// TIA Portal V20 export
DATA_BLOCK "CallEquipment_DB"   // DB148
{ DB_Accessible_From_OPC_UA := 'FALSE' }
// stored: AssignedProDiagFB Unit1.Em3.ProDiag, DBAccessibleFromOPCUA false, DBAccessibleFromWebserver false, InstanceOfName Unit1.Em3.CallEquipment, InstanceOfType FB, Namespace Unit1.Em3
"Unit1.Em3.CallEquipment"
   // VAR_INPUT
   //    ZoneOperationEnable { ExternalWritable := 'False'} : "LWONIK_typeSafetyZoneManualOperation";
   // END_VAR
   // VAR_IN_OUT
   //    unitStatus : "LAF_typeUnitStatus";
   //    emFeedback : "LUC_typeEmFeedback";
   //    unitAlarmDB : "LAF_typeAlarms";
   // END_VAR
   // VAR
   //    InstSequenceTopTapeLoading { ExternalWritable := 'False'} : "Unit1.Em3.Sequence_1_TopTapeLoading";
   //    InstSequenceTopTapeAttachment { ExternalWritable := 'False'} : "Unit1.Em3.Sequence_2_TopTapeAttachment";
   //    InstSequenceTopTapeFixStage { ExternalWritable := 'False'} : "Unit1.Em3.Sequence_3_TopTapeFixStage";
   //    instTopTapeLoadingHomeJob1 { ExternalWritable := 'False'} : "LAF_SelectJob";
   //    instTopTapeLoadingChargeJob2 { ExternalWritable := 'False'} : "LAF_SelectJob";
   //    instTopTapeAttachHomeJob1 { ExternalWritable := 'False'} : "LAF_SelectJob";
   //    instTopTapeAttachTapeGetJob2 { ExternalWritable := 'False'} : "LAF_SelectJob";
   //    instTopTapeAttachTape1PutJob3 { ExternalWritable := 'False'} : "LAF_SelectJob";
   //    instTopTapeAttachTape2PutJob4 { ExternalWritable := 'False'} : "LAF_SelectJob";
   //    instTopTapeAttachTapeIdleJob5 { ExternalWritable := 'False'} : "LAF_SelectJob";
   //    instTopTapeFixStageHomeJob1 { ExternalWritable := 'False'} : "LAF_SelectJob";
   //    instTopTapeFixStageLoadJob2 { ExternalWritable := 'False'} : "LAF_SelectJob";
   //    instTopTapeFixStageTaping1Job3 { ExternalWritable := 'False'} : "LAF_SelectJob";
   //    instTopTapeFixStageTaping2Job4 { ExternalWritable := 'False'} : "LAF_SelectJob";
   //    instTopTapeFixStageUnloadJob5 { ExternalWritable := 'False'} : "LAF_SelectJob";
   //    instCmTopTapeJRDetect { ExternalWritable := 'False'} : "LBC_DigitalSignalCn";
   //    instCmTopTapeDiameter { ExternalWritable := 'False'} : "LBC_DigitalSignalCn";
   //    instCmTopTapeAxisX { ExternalWritable := 'False'} : "LBC_Axis64Pos_TecPlcCn";
   //    instCmTopTapeAxisY { ExternalWritable := 'False'} : "LBC_Axis64Pos_TecPlcCn";
   //    instCmTopTapeLoadingFwdBwd { ExternalWritable := 'False'} : "LBC_TwoWayActuatorCn";
   //    instCmTopTapeLoadingClampOpenClose { ExternalWritable := 'False'} : "LBC_TwoWayActuatorCn";
   //    instCmTopTapeCutterUpDown { ExternalWritable := 'False'} : "LBC_TwoWayActuatorCn";
   //    instCmTopTapeCutterClampUpDown { ExternalWritable := 'False'} : "LBC_TwoWayActuatorCn";
   //    instCmTopTapeTensionFwdBwd { ExternalWritable := 'False'} : "LBC_TwoWayActuatorCn";
   //    instCmTopTapeAttachmentUpDown { ExternalWritable := 'False'} : "LBC_TwoWayActuatorCn";
   //    instCmTopTapeClampTopLeftUpDown { ExternalWritable := 'False'} : "LBC_TwoWayActuatorCn";
   //    instCmTopTapeClampTopCenterUpDown { ExternalWritable := 'False'} : "LBC_TwoWayActuatorCn";
   //    instCmTopTapeClampTopRightUpDown { ExternalWritable := 'False'} : "LBC_TwoWayActuatorCn";
   //    instCmTopTapeClampBtmDownUp { ExternalWritable := 'False'} : "LBC_TwoWayActuatorCn";
   //    instCmTopTapeClampAllOpenClose { ExternalWritable := 'False'} : "LBC_TwoWayActuatorCn";
   //    instCmTopTapeAttachmentVaccumOffOn { ExternalWritable := 'False'} : "LBC_TwoWayActuatorCn";
   //    instQrHandyReader { ExternalWritable := 'False'} : "LER_QRread_DM8700";
   //    instInterlockTopTapeAxisX { ExternalWritable := 'False'} : "LER_Axis64Pos_InterlockSummary";
   //    instInterlockTopTapeAxisY { ExternalWritable := 'False'} : "LER_Axis64Pos_InterlockSummary";
   //    instEventsPFE { ExternalWritable := 'False'} : "Unit1.Em3.EventsPFE";
   //    instManageAlarms { ExternalWritable := 'False'} : "LAF_ManageAlarms";
   //    statUnitStatus { ExternalWritable := 'False'} : "LAF_typeUnitStatus";
   //    statSlmStatus { ExternalWritable := 'False'} : Struct
   //       running : Bool;
   //       powerOff : Bool;
   //    END_STRUCT;
   //    statEmptyJobStatus { ExternalWritable := 'False'} : "LAF_typeJobStatus";
   //    statTonTime { ExternalWritable := 'False'} : Array[0..999] of TON_TIME;
   //    statTofTime { ExternalWritable := 'False'} : Array[0..9] of TOF_TIME;
   //    statPulse { ExternalWritable := 'False'} : Array[0..999] of Bool;
   //    statEnableManualCmds { ExternalWritable := 'False'} : Bool;
   //    TopTapeIdleCondition : Bool;
   //    "*** Interlock Axis ***" : Bool;
   //    TopTapeAxisX_JogCW { S7_SetPoint := 'True'} : "LER_Axis_Jog";
   //    TopTapeAxisX_JogCCW { S7_SetPoint := 'True'} : "LER_Axis_Jog";
   //    TopTapeAxisY_JogCW { S7_SetPoint := 'True'} : "LER_Axis_Jog";
   //    TopTapeAxisY_JogCCW { S7_SetPoint := 'True'} : "LER_Axis_Jog";
   //    TopTapeAxisX_interlock { S7_SetPoint := 'True'} : Array[0..10] of "LER_Axis_Absolute";
   //    TopTapeAxisY_interlock { S7_SetPoint := 'True'} : Array[0..10] of "LER_Axis_Absolute";
   //    TopTapeAxisX_IntPos : Array[0..9] of Struct
   //       "Int" : Array[1..10] of Bool;
   //    END_STRUCT;
   //    TopTapeAxisY_IntPos : Array[0..9] of Struct
   //       "Int" : Array[1..10] of Bool;
   //    END_STRUCT;
   //    TopTapeAxisX_IntHome : Array[0..9] of Bool;
   //    TopTapeAxisY_IntHome : Array[0..9] of Bool;
   //    TopTapeAxisX_PosAbsolute : Array[0..10] of Bool;
   //    TopTapeAxisY_PosAbsolute : Array[0..10] of Bool;
   //    TopTapeAxisX_Home { S7_SetPoint := 'True'} : "LER_Axis_Homing";
   //    TopTapeAxisY_Home { S7_SetPoint := 'True'} : "LER_Axis_Homing";
   //    "*** Interlock TwoWay ***" { S7_SetPoint := 'True'} : "LER_Axis_Homing";
   //    instTopTapeLoadingBwdFwdInterlock { S7_SetPoint := 'True'} : Array[0..2] of "LER_Actuator";
   //    instTopTapeLoadingClampInterlock { S7_SetPoint := 'True'} : Array[0..2] of "LER_Actuator";
   //    instTopTapeCutterUpDownInterlock { S7_SetPoint := 'True'} : Array[0..2] of "LER_Actuator";
   //    instTopTapeCutterClampInterlock { S7_SetPoint := 'True'} : Array[0..2] of "LER_Actuator";
   //    instTopTapeTensionFwdBwdInterlock { S7_SetPoint := 'True'} : Array[0..2] of "LER_Actuator";
   //    instTopTapeAttachmentUpDownInterlock { S7_SetPoint := 'True'} : Array[0..2] of "LER_Actuator";
   //    instTopTapeClampTopLeftUpDownInterlock { S7_SetPoint := 'True'} : Array[0..2] of "LER_Actuator";
   //    instTopTapeClampTopCenterUpDownInterlock { S7_SetPoint := 'True'} : Array[0..2] of "LER_Actuator";
   //    instTopTapeClampTopRightUpDownInterlock { S7_SetPoint := 'True'} : Array[0..2] of "LER_Actuator";
   //    instTopTapeClampBtmDownUpInterlock { S7_SetPoint := 'True'} : Array[0..2] of "LER_Actuator";
   //    instTopTapeClampAllOpenCloseInterlock { S7_SetPoint := 'True'} : Array[0..2] of "LER_Actuator";
   //    instTopTapeAttachmentVaccumOffOnInterlock { S7_SetPoint := 'True'} : Array[0..2] of "LER_Actuator";
   //    TopTapeLoadingBwdFwd_IntPos : Array[0..2] of Struct
   //       "Int" : Array[1..10] of Bool;
   //    END_STRUCT;
   //    TopTapeLoadingClamp_IntPos : Array[0..2] of Struct
   //       "Int" : Array[1..10] of Bool;
   //    END_STRUCT;
   //    TopTapeCutterUpDown_IntPos : Array[0..2] of Struct
   //       "Int" : Array[1..10] of Bool;
   //    END_STRUCT;
   //    TopTapeCutterClamp_IntPos : Array[0..2] of Struct
   //       "Int" : Array[1..10] of Bool;
   //    END_STRUCT;
   //    TopTapeTensionFwdBwd_IntPos : Array[0..2] of Struct
   //       "Int" : Array[1..10] of Bool;
   //    END_STRUCT;
   //    TopTapeAttachmentUpDown_IntPos : Array[0..2] of Struct
   //       "Int" : Array[1..10] of Bool;
   //    END_STRUCT;
   //    TopTapeClampTopLeftUpDown_IntPos : Array[0..2] of Struct
   //       "Int" : Array[1..10] of Bool;
   //    END_STRUCT;
   //    TopTapeClampTopCenterUpDown_IntPos : Array[0..2] of Struct
   //       "Int" : Array[1..10] of Bool;
   //    END_STRUCT;
   //    TopTapeClampTopRightUpDown_IntPos : Array[0..2] of Struct
   //       "Int" : Array[1..10] of Bool;
   //    END_STRUCT;
   //    TopTapeClampBtmDownUp_IntPos : Array[0..2] of Struct
   //       "Int" : Array[1..10] of Bool;
   //    END_STRUCT;
   //    TopTapeClampAllOpenClose_IntPos : Array[0..2] of Struct
   //       "Int" : Array[1..10] of Bool;
   //    END_STRUCT;
   //    TopTapeAttachmentVaccumOffOn_IntPos : Array[0..2] of Struct
   //       "Int" : Array[1..10] of Bool;
   //    END_STRUCT;
   //    citi_Ptrig : Array[0..20] of Bool;
   //    citiTon : Array[0..20] of TON_TIME;
   //    citi : Time;
   //    citiTest : Array[0..20] of Bool;
   // END_VAR
BEGIN
END_DATA_BLOCK
